	X =  2637.990  mm,	Y =   153.365  mm,	Z =   867.816  mm,
	W =    36.071 deg,	P =    31.153 deg,	R =     3.552 deg
   GP2:
	UF : 0, UT : 1,
	J1=    90.000 deg,	J2=   -90.000 deg
};
P[1070]{
   GP1:
	UF : 1, UT : 1,		CONFIG : 'N U T, 0, 0, 0',
	X =  2659.664  mm,	Y =   165.624  mm,	Z =  1020.932  mm,
	W =    26.374 deg,	P =    27.847 deg,	R =   -19.583 deg
   GP2:
	UF : 0, UT : 1,
	J1=    90.000 deg,	J2=   -90.000 deg
};
P[1071]{
   GP1:
	UF : 1, UT : 1,		CONFIG : 'N U T, 0, 0, 0',
	X =  2353.664  mm,	Y =    86.624  mm,	Z =   995.947  mm,
	W =    23.231 deg,	P =    35.687 deg,	R =   -21.225 deg
   GP2:
	UF : 0, UT : 1,
	J1=    90.000 deg,	J2=   -90.000 deg
};
P[1072]{
   GP1:
	UF : 1, UT : 1,		CONFIG : 'N U T, 0, 0, 0',
	X =  2347.763  mm,	Y =   140.779  mm,	Z =   874.016  mm,
	W =    23.257 deg,	P =    35.700 deg,	R =   -27.108 deg
   GP2:
	UF : 0, UT : 1,
	J1=    90.000 deg,	J2=   -90.000 deg
};
P[1073]{
   GP1:
	UF : 1, UT : 1,		CONFIG : 'N U T, 0, 0, 0',
	X =  2282.842  mm,	Y =   106.505  mm,	Z =   873.161  mm,
	W =    23.147 deg,	P =    35.649 deg,	R =   -27.171 deg
   GP2:
	UF : 0, UT : 1,
	J1=    90.000 deg,	J2=   -90.000 deg
};
P[1074]{
   GP1:
	UF : 1, UT : 1,		CONFIG : 'N U T, 0, 0, 0',
	X =  2314.873  mm,	Y =    49.882  mm,	Z =  1059.436  mm,
	W =    23.230 deg,	P =    35.687 deg,	R =   -27.122 deg
   GP2:
	UF : 0, UT : 1,
	J1=    90.000 deg,	J2=   -90.000 deg
};
P[1075]{
   GP1:
	UF : 1, UT : 1,		CONFIG : 'N U T, 0, 0, 0',
	X =  2407.391  mm,	Y =   163.912  mm,	Z =   960.657  mm,
	W =     8.539 deg,	P =    35.418 deg,	R =    39.363 deg
   GP2:
	UF : 0, UT : 1,
	J1=    90.000 deg,	J2=   -90.000 deg
};
P[1076]{
   GP1:
	UF : 1, UT : 1,		CONFIG : 'N U T, 0, 0, 0',
	X =  2350.204  mm,	Y =   145.740  mm,	Z =   875.004  mm,
	W =      .525 deg,	P =    41.703 deg,	R =    27.279 deg
   GP2:
	UF : 0, UT : 1,
	J1=    90.000 deg,	J2=   -90.000 deg
};
P[1077]{
   GP1:
	UF : 1, UT : 1,		CONFIG : 'N U T, 0, 0, 0',
	X =  2339.594  mm,	Y =   166.628  mm,	Z =   875.161  mm,
	W =      .525 deg,	P =    41.703 deg,	R =    27.279 deg
   GP2:
	UF : 0, UT : 1,
	J1=    90.000 deg,	J2=   -90.000 deg
};
P[1078]{
   GP1:
	UF : 1, UT : 1,		CONFIG : 'N U T, 0, 0, 0',
	X =  2384.166  mm,	Y =   179.687  mm,	Z =   938.550  mm,
	W =     5.309 deg,	P =    36.733 deg,	R =    27.708 deg
   GP2:
	UF : 0, UT : 1,
	J1=    90.000 deg,	J2=   -90.000 deg
};
P[1079]{
   GP1:
	UF : 1, UT : 1,		CONFIG : 'N U T, 0, 0, 0',
	X =  2240.873  mm,	Y =   177.882  mm,	Z =  1059.436  mm,
	W =   -27.572 deg,	P =    24.023 deg,	R =    68.377 deg
   GP2:
	UF : 0, UT : 1,
	J1=    90.000 deg,	J2=   -90.000 deg
};
P[1080]{
   GP1:
	UF : 1, UT : 1,		CONFIG : 'N U T, 0, 0, 0',
	X =  2266.854  mm,	Y =   128.932  mm,	Z =   873.962  mm,
	W =   -30.363 deg,	P =    30.099 deg,	R =    67.112 deg
   GP2:
	UF : 0, UT : 1,
	J1=    90.000 deg,	J2=   -90.000 deg
};
P[1081]{
   GP1:
	UF : 1, UT : 1,		CONFIG : 'N U T, 0, 0, 0',
	X =  2329.302  mm,	Y =   165.062  mm,	Z =   875.549  mm,
	W =   -30.345 deg,	P =    30.078 deg,	R =    67.107 deg
   GP2:
	UF : 0, UT : 1,
	J1=    90.000 deg,	J2=   -90.000 deg
};
P[1082]{
   GP1:
	UF : 1, UT : 1,		CONFIG : 'N U T, 0, 0, 0',
	X =  2295.490  mm,	Y =   194.983  mm,	Z =   940.815  mm,
	W =   -30.368 deg,	P =    30.111 deg,	R =    93.411 deg
   GP2:
	UF : 0, UT : 1,
	J1=    90.000 deg,	J2=   -90.000 deg
};
P[1083]{
   GP1:
	UF : 1, UT : 1,		CONFIG : 'N U T, 0, 0, 0',
	X =  2098.039  mm,	Y =    95.390  mm,	Z =  1058.670  mm,
	W =    -8.223 deg,	P =    27.055 deg,	R =    52.392 deg
   GP2:
	UF : 0, UT : 1,
	J1=    90.000 deg,	J2=   -90.000 deg
};
P[1084]{
   GP1:
	UF : 1, UT : 1,		CONFIG : 'N U T, 0, 0, 0',
	X =  1658.214  mm,	Y =    44.710  mm,	Z =   967.832  mm,
	W =    -2.274 deg,	P =    43.564 deg,	R =   -25.102 deg
   GP2:
	UF : 0, UT : 1,
	J1=    90.000 deg,	J2=   -90.000 deg
};
P[1085]{
   GP1:
	UF : 1, UT : 1,		CONFIG : 'N U T, 0, 0, 0',
	X =  1616.012  mm,	Y =    61.843  mm,	Z =   869.524  mm,
	W =    -2.210 deg,	P =    43.585 deg,	R =   -25.052 deg
   GP2:
	UF : 0, UT : 1,
	J1=    90.000 deg,	J2=   -90.000 deg
};
P[1086]{
   GP1:
	UF : 1, UT : 1,		CONFIG : 'N U T, 0, 0, 0',
	X =  1672.594  mm,	Y =   479.618  mm,	Z =   872.893  mm,
	W =    39.799 deg,	P =    19.526 deg,	R =    46.352 deg
   GP2:
	UF : 0, UT : 1,
	J1=    90.000 deg,	J2=   -90.000 deg
};
P[1087]{
   GP1:
	UF : 1, UT : 1,		CONFIG : 'N U T, 0, 0, 0',
	X =  1706.217  mm,	Y =   503.296  mm,	Z =   954.723  mm,
	W =    37.796 deg,	P =     8.495 deg,	R =    37.859 deg
   GP2:
	UF : 0, UT : 1,
	J1=    90.000 deg,	J2=   -90.000 deg
};
P[1088]{
   GP1:
	UF : 1, UT : 1,		CONFIG : 'N U T, 0, 0, 0',
	X =  1481.499  mm,	Y =    22.372  mm,	Z =  1018.721  mm,
	W =    -2.274 deg,	P =    43.564 deg,	R =  -148.737 deg
   GP2:
	UF : 0, UT : 1,
	J1=    90.000 deg,	J2=   -90.000 deg
};
P[1089]{
   GP1:
	UF : 1, UT : 1,		CONFIG : 'N U T, 0, 0, -1',
	X =  1598.141  mm,	Y =    61.873  mm,	Z =   868.998  mm,
	W =    -2.313 deg,	P =    43.575 deg,	R =   179.472 deg
   GP2:
	UF : 0, UT : 1,
	J1=    90.000 deg,	J2=   -90.000 deg
};
P[1090]{
   GP1:
	UF : 1, UT : 1,		CONFIG : 'N U T, 0, 0, -1',
	X =  1654.326  mm,	Y =   474.279  mm,	Z =   873.521  mm,
	W =   -36.221 deg,	P =    26.164 deg,	R =   127.253 deg
   GP2:
	UF : 0, UT : 1,
	J1=    90.000 deg,	J2=   -90.000 deg
};
P[1091]{
   GP1:
	UF : 1, UT : 1,		CONFIG : 'N U T, 0, 0, -1',
	X =  1571.244  mm,	Y =   480.285  mm,	Z =   955.523  mm,
	W =   -38.018 deg,	P =    23.214 deg,	R =   151.318 deg
   GP2:
	UF : 0, UT : 1,
	J1=    90.000 deg,	J2=   -90.000 deg
};
P[1092]{
   GP1:
	UF : 1, UT : 1,		CONFIG : 'N U T, 0, 0, 0',
	X =  1635.521  mm,	Y =   132.162  mm,	Z =  1231.477  mm,
	W =    25.682 deg,	P =    77.887 deg,	R =   -93.023 deg
   GP2:
	UF : 0, UT : 1,
	J1=    90.000 deg,	J2=   -90.000 deg
};
P[1093]{
   GP1:
	UF : 1, UT : 1,		CONFIG : 'N U T, 0, 0, 0',
	X =  1143.065  mm,	Y = -1469.733  mm,	Z =  1613.189  mm,
	W =   -45.551 deg,	P =   -20.029 deg,	R =   -44.051 deg
   GP2:
	UF : 0, UT : 1,
	J1=    90.000 deg,	J2=   -80.000 deg
};
P[1094]{
   GP1:
	UF : 1, UT : 1,		CONFIG : 'F U T, 0, 0, 0',
	X =  2542.229  mm,	Y = -1549.271  mm,	Z =  1152.755  mm,
	W =   -35.769 deg,	P =   -28.014 deg,	R =    20.274 deg
   GP2:
	UF : 0, UT : 1,
	J1=    90.000 deg,	J2=   -80.000 deg
};
P[1095]{
   GP1:
	UF : 1, UT : 1,		CONFIG : 'F U T, 0, 0, 0',
	X =  2483.627  mm,	Y = -1623.804  mm,	Z =   973.832  mm,
	W =   -35.088 deg,	P =   -31.677 deg,	R =    63.073 deg
   GP2:
	UF : 0, UT : 1,
	J1=    90.000 deg,	J2=   -80.000 deg
};
P[1096]{
   GP1:
	UF : 1, UT : 1,		CONFIG : 'F U T, 0, 0, 0',
	X =  2752.122  mm,	Y = -1559.636  mm,	Z =   709.416  mm,
	W =   -35.088 deg,	P =   -31.677 deg,	R =    63.073 deg
   GP2:
	UF : 0, UT : 1,
	J1=    90.000 deg,	J2=   -80.000 deg
};
P[1097]{
   GP1:
	UF : 1, UT : 1,		CONFIG : 'F U T, 0, 0, 0',
	X =  2857.673  mm,	Y = -1474.003  mm,	Z =   621.464  mm,
	W =   -15.693 deg,	P =   -49.080 deg,	R =    48.928 deg
   GP2:
	UF : 0, UT : 1,
	J1=    89.999 deg,	J2=   -80.000 deg
};
P[1098]{
   GP1:
	UF : 1, UT : 1,		CONFIG : 'F U T, 0, 0, 0',
	X =  2861.892  mm,	Y = -1519.562  mm,	Z =   611.305  mm,
	W =   -25.979 deg,	P =   -39.192 deg,	R =    47.476 deg
   GP2:
	UF : 0, UT : 1,
	J1=    90.000 deg,	J2=   -80.000 deg
};
P[1099]{
   GP1:
	UF : 1, UT : 1,		CONFIG : 'F U T, 0, 0, 0',
	X =  2849.490  mm,	Y = -1550.087  mm,	Z =   609.269  mm,
	W =   -35.101 deg,	P =   -20.655 deg,	R =    48.398 deg
   GP2:
	UF : 0, UT : 1,
	J1=    90.000 deg,	J2=   -80.000 deg
};
P[1100]{
   GP1:
	UF : 1, UT : 1,		CONFIG : 'F U T, 0, 0, 0',
	X =  2829.027  mm,	Y = -1574.688  mm,	Z =   602.044  mm,
	W =   -35.568 deg,	P =   -11.954 deg,	R =    36.091 deg
   GP2:
	UF : 0, UT : 1,
	J1=    90.000 deg,	J2=   -80.000 deg
};
P[1101]{
   GP1:
	UF : 1, UT : 1,		CONFIG : 'F U T, 0, 0, 0',
	X =  2761.067  mm,	Y = -1614.938  mm,	Z =   596.786  mm,
	W =   -35.568 deg,	P =   -11.953 deg,	R =    36.091 deg
   GP2:
	UF : 0, UT : 1,
	J1=    90.000 deg,	J2=   -80.000 deg
};
P[1102]{
   GP1:
	UF : 1, UT : 1,		CONFIG : 'F U T, 0, 0, 0',
	X =  2698.117  mm,	Y = -1568.160  mm,	Z =   671.710  mm,
	W =   -43.039 deg,	P =   -10.740 deg,	R =    31.361 deg
   GP2:
	UF : 0, UT : 1,
	J1=    90.000 deg,	J2=   -80.000 deg
};
P[1103]{
   GP1:
	UF : 1, UT : 1,		CONFIG : 'F U T, 0, 0, 0',
	X =  2600.787  mm,	Y = -1658.895  mm,	Z =   858.622  mm,
	W =  -106.889 deg,	P =    58.736 deg,	R =    44.006 deg
   GP2:
	UF : 0, UT : 1,
	J1=    90.000 deg,	J2=   -80.000 deg
};
P[1104]{
   GP1:
	UF : 1, UT : 1,		CONFIG : 'F U T, 0, 0, 0',
	X =  2649.433  mm,	Y = -1667.474  mm,	Z =   680.642  mm,
	W =    47.958 deg,	P =    12.926 deg,	R =   -63.288 deg
   GP2:
	UF : 0, UT : 1,
	J1=    90.000 deg,	J2=   -80.000 deg
};
P[1105]{
   GP1:
	UF : 1, UT : 1,		CONFIG : 'F U T, 0, 0, 0',
	X =  2764.132  mm,	Y = -1619.624  mm,	Z =   592.114  mm,
	W =    49.127 deg,	P =    13.962 deg,	R =   -64.233 deg
   GP2:
	UF : 0, UT : 1,
	J1=    90.000 deg,	J2=   -80.000 deg
};
P[1106]{
   GP1:
	UF : 1, UT : 1,		CONFIG : 'F U T, 0, 0, 0',
	X =  2777.012  mm,	Y = -1644.965  mm,	Z =   588.867  mm,
	W =    49.101 deg,	P =    13.947 deg,	R =   -64.231 deg
   GP2:
	UF : 0, UT : 1,
	J1=    90.000 deg,	J2=   -80.000 deg
};
P[1107]{
   GP1:
	UF : 1, UT : 1,		CONFIG : 'F U T, 0, 0, 0',
	X =  2707.461  mm,	Y = -1664.975  mm,	Z =   637.599  mm,
	W =    48.076 deg,	P =     9.473 deg,	R =   -69.425 deg
   GP2:
	UF : 0, UT : 1,
	J1=    90.000 deg,	J2=   -80.000 deg
};
P[1108]{
   GP1:
	UF : 1, UT : 1,		CONFIG : 'F U T, 0, 0, 0',
	X =  2438.792  mm,	Y = -1806.240  mm,	Z =  1074.483  mm,
	W =    50.396 deg,	P =     5.479 deg,	R =   -69.123 deg
   GP2:
	UF : 0, UT : 1,
	J1=    90.000 deg,	J2=   -80.000 deg
};
P[1109]{
   GP1:
	UF : 1, UT : 1,		CONFIG : 'F U T, 0, 0, 0',
	X =  1894.275  mm,	Y = -1518.285  mm,	Z =  2086.944  mm,
	W =    58.754 deg,	P =   -40.157 deg,	R =   -73.858 deg
   GP2:
	UF : 0, UT : 1,
	J1=    90.000 deg,	J2=   -80.000 deg
};
P[1110]{
   GP1:
	UF : 1, UT : 1,		CONFIG : 'N U B, 0, 0, 0',
	X =   390.531  mm,	Y =    -9.911  mm,	Z =  2433.853  mm,
	W =     -.021 deg,	P =   -39.773 deg,	R =      .020 deg
   GP2:
	UF : 0, UT : 1,
	J1=    90.000 deg,	J2=   -80.000 deg
};
P[1111]{
   GP1:
	UF : 1, UT : 1,
	J1=     7.148 deg,	J2=   -36.542 deg,	J3=    36.380 deg,
	J4=   -17.109 deg,	J5=   -53.805 deg,	J6=    12.574 deg
   GP2:
	UF : 0, UT : 1,
	J1=    90.000 deg,	J2=  -135.000 deg
};
P[1112]{
   GP1:
	UF : 1, UT : 1,		CONFIG : 'N U T, 0, 0, 0',
	X =  2113.870  mm,	Y =   780.736  mm,	Z =   928.722  mm,
	W =    12.771 deg,	P =   -18.901 deg,	R =    28.710 deg
   GP2:
	UF : 0, UT : 1,
	J1=    90.000 deg,	J2=  -135.000 deg
};
P[1113]{
   GP1:
	UF : 1, UT : 1,		CONFIG : 'N U T, 0, 0, 0',
	X =  2397.681  mm,	Y =   841.473  mm,	Z =   828.772  mm,
	W =    12.771 deg,	P =   -18.901 deg,	R =    28.710 deg
   GP2:
	UF : 0, UT : 1,
	J1=    90.000 deg,	J2=  -135.000 deg
};
P[1114]{
   GP1:
	UF : 1, UT : 1,		CONFIG : 'N U T, 0, 0, 0',
	X =  2651.304  mm,	Y =  1015.539  mm,	Z =   531.056  mm,
	W =    12.771 deg,	P =   -18.901 deg,	R =    55.019 deg
   GP2:
	UF : 0, UT : 1,
	J1=    90.000 deg,	J2=  -135.000 deg
};
P[1115]{
   GP1:
	UF : 1, UT : 1,		CONFIG : 'N U T, 0, 0, 0',
	X =  2648.832  mm,	Y =  1039.517  mm,	Z =   445.697  mm,
	W =     2.946 deg,	P =    -4.536 deg,	R =    57.038 deg
   GP2:
	UF : 0, UT : 1,
	J1=    90.000 deg,	J2=  -135.000 deg
};
P[1116]{
   GP1:
	UF : 1, UT : 1,		CONFIG : 'N U T, 0, 0, 0',
	X =  2677.404  mm,	Y =  1039.517  mm,	Z =   445.698  mm,
	W =     2.946 deg,	P =    -4.536 deg,	R =    57.038 deg
   GP2:
	UF : 0, UT : 1,
	J1=    90.000 deg,	J2=  -135.000 deg
};
P[1117]{
   GP1:
	UF : 1, UT : 1,		CONFIG : 'N U T, 0, 0, 0',
	X =  2651.304  mm,	Y =  1015.539  mm,	Z =   531.056  mm,
	W =    12.771 deg,	P =   -18.901 deg,	R =    55.019 deg
   GP2:
	UF : 0, UT : 1,
	J1=    90.000 deg,	J2=  -135.000 deg
};
P[1118]{
   GP1:
	UF : 1, UT : 1,		CONFIG : 'N U T, 0, 0, 0',
	X =  2397.681  mm,	Y =   841.473  mm,	Z =   828.772  mm,
	W =    12.771 deg,	P =   -18.901 deg,	R =    28.710 deg
   GP2:
	UF : 0, UT : 1,
	J1=    90.000 deg,	J2=  -135.000 deg
};
P[1119]{
   GP1:
	UF : 1, UT : 1,		CONFIG : 'N U T, 0, 0, 0',
	X =  1853.840  mm,	Y =   735.295  mm,	Z =  1070.725  mm,
	W =    12.871 deg,	P =   -19.018 deg,	R =    29.278 deg
   GP2:
	UF : 0, UT : 1,
	J1=    90.000 deg,	J2=  -135.000 deg
};
/END
